//==================================================================================================
//							Beckhoff Automation Poland
//									23.05.2018
//	Blok zmienia stan EtherCAT Slave i monitoruje flage ukonczenia
//
//	Niezbedne biblioteki: Tc2_EtherCAT
//
// 	v1.1	|| TC v 3.1.4022.16	|| - optymalizacja kodu
// 	v1.0	|| TC v 3.1.4020.32	|| - pierwsza wersja
//==================================================================================================
FUNCTION_BLOCK FB_ChangeEtherCATSlaveState
VAR_INPUT
	bExecute								: BOOL;							// Start on rising edge
	sEtherCAT_NetID							: STRING;						// EtherCAT Master NetID
	nSlaveAddr								: UINT;							// EtherCAT Drive slave port
	byReguestedState						: BYTE;							(* 	16#1- EC_DEVICE_STATE_INIT  
																				16#2- EC_DEVICE_STATE_PREOP     
																				16#3- EC_DEVICE_STATE_BOOTSTRAP     
																				16#4- EC_DEVICE_STATE_SAFEOP  
																				16#8- EC_DEVICE_STATE_OP
																				16#10- EC_DEVICE_STATE_ERROR  *)
END_VAR
VAR_OUTPUT
	byActualState							: BYTE;							(* 	16#1-EC_DEVICE_STATE_INIT  
																				16#2-EC_DEVICE_STATE_PREOP     
																				16#3-EC_DEVICE_STATE_BOOTSTRAP     
																				16#4-EC_DEVICE_STATE_SAFEOP  
																				16#8-EC_DEVICE_STATE_OP
																				16#10-EC_DEVICE_STATE_ERROR  *)
	bBusy									: BOOL;
	bDone									: BOOL;
	bError									: BOOL;
	udiErrorID								: UDINT;	
END_VAR
VAR	
	fbEcReqSlaveState						: FB_EcReqSlaveState;
	fbEcGetSlaveState						: FB_EcGetSlaveState;
	timerTON								: TON;
	rtExecute								: R_TRIG;
	iState									: INT;
	iTry									: INT;							// number of tries
END_VAR

timerTON(PT:=T#500MS);
rtExecute(CLK:=bExecute);

CASE iState OF

	0:																// Init parameters
		IF rtExecute.Q THEN
			bBusy							:= TRUE;
			bDone							:= FALSE;
			bError							:= FALSE;
			udiErrorID						:= 0;
			iTry							:= 0;
			fbEcReqSlaveState.sNetId		:= sEtherCAT_NetID; 
			fbEcGetSlaveState.sNetId		:= sEtherCAT_NetID; 
			fbEcReqSlaveState.nSlaveAddr	:= nSlaveAddr; 
			fbEcGetSlaveState.nSlaveAddr	:= nSlaveAddr;
			fbEcReqSlaveState.state			:= byReguestedState;
			fbEcReqSlaveState.bExecute		:= TRUE;
			iState							:= iState + 10;			
		END_IF
		
	10:																// State request
		fbEcReqSlaveState.bExecute			:= FALSE;
		IF NOT fbEcReqSlaveState.bBusy THEN
			IF fbEcReqSlaveState.bError THEN
				iState						:= 99;
			ELSE
				iState						:= iState + 10;
			END_IF
		END_IF

		
	20:																// Request every 0.5s
		timerTON.IN							:= TRUE;
		IF timerTON.Q THEN
			timerTON.IN						:= FALSE;
			fbEcGetSlaveState.bExecute		:= TRUE;
			iState							:= iState + 10;
		END_IF
		
	30:																// Done already?
		fbEcGetSlaveState.bExecute			:= FALSE;	
		IF NOT fbEcGetSlaveState.bBusy THEN
			IF NOT fbEcGetSlaveState.bError AND fbEcGetSlaveState.state.deviceState = fbEcReqSlaveState.state THEN
				bBusy						:= FALSE;
				bDone						:= TRUE;
				iState						:= 0;
			ELSIF iTry = 40 THEN
				iState						:= 99;
			ELSE
				iTry						:= iTry + 1;
				iState						:= iState - 10;			
			END_IF
			byActualState					:= fbEcGetSlaveState.state.deviceState;
		END_IF
		
	99:																// ERROR STATE
		bError 								:= TRUE;
		bBusy								:= FALSE;
		udiErrorID							:= fbEcReqSlaveState.nErrId + fbEcGetSlaveState.nErrId;
		iState								:= 0;
		
END_CASE

fbEcReqSlaveState();
fbEcGetSlaveState();

END_FUNCTION_BLOCK

(* stored: Version 1.1.0.1, ProductVersion 3.1.4026.13, FileIdentifier 8a6fa5dd7b1ac168c209f42ec5d4e1e84a525e17, FileSignature a27b363007b387fa1a77486772403f94adad133bed8c40f428a0cc2a3a74ba554fc05a8ffcb671bd9e938e10c8400bf0ea77ed3a4e4cc10c46d3bc6cfd1cbad302199460f3b9dfbaa408067ccb044ce987ce2f5c34b2e553bf6cb30e8dfece9099d0a3a84fe5cadb366a3b43125a8ba56d943c58d37b4fa6a6b50890a9bce5dda9e4e593554accbc90f802c11af0f1e7f18025fa288cb5909a7c0c6ce411c9e17159d22e59716fe306a7e6c9dbf60c1698208f71ab650cb9c03049e3cef45ac7010057480899f4dca8c3fcdb26ca06ceb5fa26a53a62d031e045e8aba08722ff0027fb3807a132764ddeaa061512400431431bcfd48a210180fb17b23e59cb39
   POU FB_ChangeEtherCATSlaveState: Id {64311408-f2d2-4d7b-a037-fcc411662873}, SpecialFunc None *)
